(* IEC 61131-3 sources: AXOpen/src/integrations/app/src/Examples/AXOpen.AxoSequencerContainer, 2 files *)

(* ---- AxoSequencerContainerDocuExample.st ---- *)
USING AXOpen.Core;

NAMESPACE AxoSequencerContainerExamples
    {S7.extern=ReadWrite}
    CLASS AxoSequencerContainerDocuExample EXTENDS  AXOpen.Core.AxoSequencerContainer
        VAR PUBLIC
            _step_1 : AxoStep;
            _step_2 : AxoStep;
            _step_3 : AxoStep;
            _myCounter : ULINT;
        END_VAR
        //<MAIN>
        METHOD PROTECTED OVERRIDE MAIN
            _myCounter := _myCounter + ULINT#1;

            IF(_step_1.Execute(THIS)) THEN
                IF(_myCounter >= ULINT#100 ) THEN
                    _myCounter := ULINT#0;
                    THIS.MoveNext();
                END_IF;
            END_IF;

            IF(_step_2.Execute(THIS)) THEN
                IF(_myCounter >= ULINT#100) THEN
                    _myCounter := ULINT#0;
                    THIS.MoveNext();
                END_IF;
            END_IF;

            IF(_step_3.Execute(THIS)) THEN
                IF(_myCounter >= ULINT#100) THEN
                    _myCounter := ULINT#0;
                    _step_3.ThrowWhen(TRUE);
                    THIS.CompleteSequence();
                END_IF;
            END_IF;
        END_METHOD
        //</MAIN>
    END_CLASS

    {S7.extern=ReadWrite}
    CLASS AxoSequencerContainerContext EXTENDS  AXOpen.Core.AxoContext
        //<InstanceDeclaration>
        VAR PUBLIC
            _mySequencerContainer : AxoSequencerContainerDocuExample;
            _rootObject : AxoObject;
        END_VAR
        //</InstanceDeclaration>

        METHOD PROTECTED OVERRIDE Main
            THIS.InitializeRootObject(_rootObject);
            //<InstanceRunning>
            _mySequencerContainer.Run(_rootObject);
            //</InstanceRunning>
        END_METHOD

    END_CLASS
END_NAMESPACE

(* ---- AxoSequencerContainerExample.st ---- *)
USING AXOpen.Core;

NAMESPACE AxoSequencerContainerExamples

    {S7.extern=ReadWrite}
    CLASS AxoSequencerContainerExample EXTENDS AXOpen.Core.AxoSequencerContainer

        VAR PUBLIC
            Counter : ULINT;
            {#ix-set:Description = "Step number one"}
            step_1 : AxoStep;
            {#ix-set:Description = "Step number two"}
            step_2 : AxoStep;
            {#ix-set:Description = "Step number three"}
            step_3 : AxoStep;
            {#ix-set:Description = "Step number four"}
            step_4 : AxoStep;
            {#ix-set:Description = "Step number five"}
            step_5 : AxoStep;
            {#ix-set:Description = "Step number six"}
            step_6 : AxoStep;
            {#ix-set:Description = "Step number seven"}
            step_7 : AxoStep;
            {#ix-set:Description = "Step number eight"}
            step_8 : AxoStep;
            {#ix-set:Description = "Step number nine"}
            step_9 : AxoStep;
            {#ix-set:Description = "Step number ten"}
            step_10 : AxoStep;
        END_VAR

        METHOD PROTECTED OVERRIDE Main

            Counter := Counter + ULINT#1;

            IF(step_1.Execute(THIS)) THEN
                IF(Counter >= ULINT#100 ) THEN
                    Counter := ULINT#0;
                    THIS.MoveNext();
                END_IF;
            END_IF;

            IF(step_2.Execute(THIS)) THEN
                IF(Counter >= ULINT#100) THEN
                    Counter := ULINT#0;
                END_IF;
            END_IF;

            IF(step_3.Execute(THIS)) THEN
                IF(Counter >= ULINT#100) THEN
                    Counter := ULINT#0;
                    step_3.ThrowWhen(TRUE);
                    THIS.MoveNext();
                END_IF;
            END_IF;

            IF(step_4.Execute(THIS)) THEN
                IF(Counter >= ULINT#100) THEN
                    Counter := ULINT#0;
                    THIS.MoveNext();
                END_IF;
            END_IF;

            IF(step_5.Execute(THIS)) THEN
                IF(Counter >= ULINT#100) THEN
                    Counter := ULINT#0;
                    THIS.MoveNext();
                END_IF;
            END_IF;

            IF(step_6.Execute(THIS)) THEN
                IF(Counter >= ULINT#100) THEN
                    Counter := ULINT#0;
                    THIS.MoveNext();
                END_IF;
            END_IF;

            IF(step_7.Execute(THIS)) THEN
                IF(Counter >= ULINT#100) THEN
                    Counter := ULINT#0;
                    THIS.MoveNext();
                END_IF;
            END_IF;

            IF(step_8.Execute(THIS)) THEN
                IF(Counter >= ULINT#100) THEN
                    Counter := ULINT#0;
                    THIS.MoveNext();
                END_IF;
            END_IF;

            IF(step_9.Execute(THIS)) THEN
                IF(Counter >= ULINT#100) THEN
                    Counter := ULINT#0;
                    THIS.MoveNext();
                END_IF;
            END_IF;

            IF(step_10.Execute(THIS)) THEN
                IF(Counter >= ULINT#100) THEN
                    Counter := ULINT#0;
                    THIS.CompleteSequence();
                END_IF;
            END_IF;
        END_METHOD
    END_CLASS

    {S7.extern=ReadWrite}
    CLASS SequencerContainerExample EXTENDS  AXOpen.Core.AxoContext
        VAR PUBLIC
            {#ix-set:AttributeName = "<#Sequencer container example#>"}
            _SequencerContainerExample : AxoSequencerContainerExample;
            _rootObject : AxoObject;
        END_VAR

        METHOD PROTECTED OVERRIDE Main
            THIS.InitializeRootObject(_rootObject);
            _SequencerContainerExample.Run(_rootObject);
        END_METHOD
    END_CLASS
END_NAMESPACE
